PROGRAM P_CraneControl
VAR
	fbTime		:	FB_Clock;
	fbSetMode	:	FB_SetMode;
	eMode 		:	E_Mode;
	
END_VAR



fbTime
(
	bStart := G_Input.bStartSwitch,
	bStop := G_Input.bStopSwitch,
	fCycleTime := G_Parameter.fCycleTime,
	fTimeInSeconds => G_Parameter.fTime
	
);
	
fbSetMode
(
	bPower := G_Input.bPoweSwitch,
	bOn := G_Input.bOnOffSwitch,
	bMode := G_Input.bModeSwitch,
	bStart := G_Input.bStartSwitch,
	bStop := G_Input.bStopSwitch,
	eMode => G_Parameter.eMode,
	bGreenLight => G_Output.bGreenLed,
	bRedLight => G_Output.bRedLed,
	sMode => G_Output.sModeDisplay	
);


IF G_Input.bPoweSwitch = FALSE OR G_Input.bOnOffSwitch = FALSE OR G_Input.bStopSwitch = TRUE THEN
	G_Input.bStartSwitch := FALSE;
	G_Input.bStopSwitch := FALSE;
END_IF

END_PROGRAM

(* stored: Version 1.1.0.1, ProductVersion 3.1.4024.10
   POU P_CraneControl: Id {a9f0b871-a372-4028-9baa-1603f14d2aaa}, SpecialFunc None *)
